(* IEC 61131-3 sources: com.logicals.lc3.webinar/usRTS_RPMControl_iSOC/src_FB_LIB_SAFE/Numeric/LINT, 8 files *)

(* ---- wADD_LINT_2.iecst ---- *)
NAMESPACE logicals.web.standard
NAMESPACE numeric

/*
 * Function block wrapper for IEC 61131-3 ADD<br>
 * IN1 =  1st value (LINT)<br>
 * IN2 =  2nd value (LINT)<br>
 * OUT = Sum of all input values (LINT)<br>
 */
FUNCTION_BLOCK wADD_LINT_2
	{ vNameAlignment:="center"; altName:="+"; bgColor:="LightPink"; width:=40; hideIONames; }
	VAR_INPUT
		IN1 : LINT;
		IN2 : LINT;
	END_VAR
	VAR_OUTPUT
		OUT : LINT;
	END_VAR

	OUT := ADD(IN1:=IN1, IN2:=IN2, ENO=>ENO);
END_FUNCTION_BLOCK

END_NAMESPACE
END_NAMESPACE

(* ---- wADD_LINT_3.iecst ---- *)
NAMESPACE logicals.web.standard
NAMESPACE numeric

/*
 * Function block wrapper for IEC 61131-3 ADD<br>
 * IN1 =  1st value (LINT)<br>
 * IN2 =  2nd value (LINT)<br>
 * IN3 =  3rd value (LINT)<br>
 * OUT = Sum of all input values (LINT)<br>
 */
FUNCTION_BLOCK wADD_LINT_3
	{ vNameAlignment:="center"; altName:="+"; bgColor:="LightPink"; width:=40; hideIONames; }
	VAR_INPUT
		IN1 : LINT;
		IN2 : LINT;
		IN3 : LINT;
	END_VAR
	VAR_OUTPUT
		OUT : LINT;
	END_VAR

	OUT := ADD(IN1:=IN1, IN2:=IN2, IN3:=IN3, ENO=>ENO);
END_FUNCTION_BLOCK

END_NAMESPACE
END_NAMESPACE

(* ---- wADD_LINT_4.iecst ---- *)
NAMESPACE logicals.web.standard
NAMESPACE numeric

/*
 * Function block wrapper for IEC 61131-3 ADD<br>
 * IN1 =  1st value (LINT)<br>
 * IN2 =  2nd value (LINT)<br>
 * IN3 =  3rd value (LINT)<br>
 * IN4 =  4th value (LINT)<br>
 * OUT = Sum of all input values (LINT)<br>
 */
FUNCTION_BLOCK wADD_LINT_4
	{ vNameAlignment:="center"; altName:="+"; bgColor:="LightPink"; width:=40; hideIONames; }
	VAR_INPUT
		IN1 : LINT;
		IN2 : LINT;
		IN3 : LINT;
		IN4 : LINT;
	END_VAR
	VAR_OUTPUT
		OUT : LINT;
	END_VAR

	OUT := ADD(IN1:=IN1, IN2:=IN2, IN3:=IN3, IN4:=IN4, ENO=>ENO);
END_FUNCTION_BLOCK

END_NAMESPACE
END_NAMESPACE

(* ---- wDIV_LINT.iecst ---- *)
NAMESPACE logicals.web.standard
NAMESPACE numeric

/*
 * Function block wrapper for IEC 61131-3 DIV<br>
 * IN1 =  1st value (LINT)<br>
 * IN2 =  2nd value (LINT)<br>
 * OUT = quotient of IN1 divided by IN2 (LINT)<br>
 */
FUNCTION_BLOCK wDIV_LINT
	{ vNameAlignment:="center"; altName:="/"; bgColor:="LightPink"; width:=40; hideIONames; }
	VAR_INPUT
		IN1 : LINT;
		IN2 : LINT;
	END_VAR
	VAR_OUTPUT
		OUT : LINT;
	END_VAR

	OUT := DIV(IN1:=IN1, IN2:=IN2, ENO=>ENO);
END_FUNCTION_BLOCK

END_NAMESPACE
END_NAMESPACE

(* ---- wMUL_LINT_2.iecst ---- *)
NAMESPACE logicals.web.standard
NAMESPACE numeric

/*
 * Function block wrapper for IEC 61131-3 MUL<br>
 * IN1 =  1st value (LINT)<br>
 * IN2 =  2nd value (LINT)<br>
 * OUT = Product of multiplication of all inputs (LINT)<br>
 */
FUNCTION_BLOCK wMUL_LINT_2
	{ vNameAlignment:="center"; altName:="*"; bgColor:="LightPink"; width:=40; hideIONames; }
	VAR_INPUT
		IN1 : LINT;
		IN2 : LINT;
	END_VAR
	VAR_OUTPUT
		OUT : LINT;
	END_VAR

	OUT := MUL(IN1:=IN1, IN2:=IN2, ENO=>ENO);
END_FUNCTION_BLOCK

END_NAMESPACE
END_NAMESPACE

(* ---- wMUL_LINT_3.iecst ---- *)
NAMESPACE logicals.web.standard
NAMESPACE numeric

/*
 * Function block wrapper for IEC 61131-3 MUL<br>
 * IN1 =  1st value (LINT)<br>
 * IN2 =  2nd value (LINT)<br>
 * IN3 =  3rd value (LINT)<br>
 * OUT = Product of multiplication of all inputs (LINT)<br>
 */
FUNCTION_BLOCK wMUL_LINT_3
	{ vNameAlignment:="center"; altName:="*"; bgColor:="LightPink"; width:=40; hideIONames; }
	VAR_INPUT
		IN1 : LINT;
		IN2 : LINT;
		IN3 : LINT;
	END_VAR
	VAR_OUTPUT
		OUT : LINT;
	END_VAR

	OUT := MUL(IN1:=IN1, IN2:=IN2, IN3:=IN3, ENO=>ENO);
END_FUNCTION_BLOCK

END_NAMESPACE
END_NAMESPACE

(* ---- wMUL_LINT_4.iecst ---- *)
NAMESPACE logicals.web.standard
NAMESPACE numeric

/*
 * Function block wrapper for IEC 61131-3 MUL<br>
 * IN1 =  1st value (LINT)<br>
 * IN2 =  2nd value (LINT)<br>
 * IN3 =  3rd value (LINT)<br>
 * IN4 =  4th value (LINT)<br>
 * OUT = Product of multiplication of all inputs (LINT)<br>
 */
FUNCTION_BLOCK wMUL_LINT_4
	{ vNameAlignment:="center"; altName:="*"; bgColor:="LightPink"; width:=40; hideIONames; }
	VAR_INPUT
		IN1 : LINT;
		IN2 : LINT;
		IN3 : LINT;
		IN4 : LINT;
	END_VAR
	VAR_OUTPUT
		OUT : LINT;
	END_VAR

	OUT := MUL(IN1:=IN1, IN2:=IN2, IN3:=IN3, IN4:=IN4, ENO=>ENO);
END_FUNCTION_BLOCK

END_NAMESPACE
END_NAMESPACE

(* ---- wSUB_LINT.iecst ---- *)
NAMESPACE logicals.web.standard
NAMESPACE numeric

/*
 * Function block wrapper for IEC 61131-3 SUB<br>
 * IN1 =  1st value (LINT)<br>
 * IN2 =  2nd value (LINT)<br>
 * OUT = IN1 minus IN2 (LINT)<br>
 */
FUNCTION_BLOCK wSUB_LINT
	{ vNameAlignment:="center"; altName:="-"; bgColor:="LightPink"; width:=40; hideIONames; }
	VAR_INPUT
		IN1 : LINT;
		IN2 : LINT;
	END_VAR
	VAR_OUTPUT
		OUT : LINT;
	END_VAR

	OUT := SUB(IN1:=IN1, IN2:=IN2, ENO=>ENO);
END_FUNCTION_BLOCK

END_NAMESPACE
END_NAMESPACE
